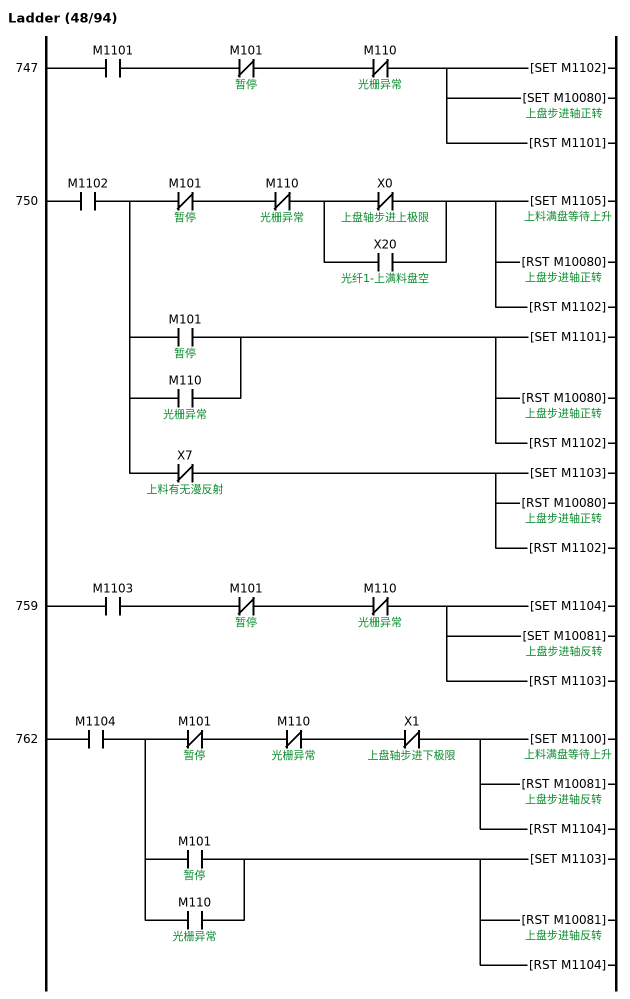
[picture p48: Ladder rows 747-762]
LD     M1101
ANI    M101	; 暂停
ANI    M110	; 光栅异常
SET    M1102
SET    M10080	; 上盘步进轴正转
RST    M1101
LD     M1102
MPS
ANI    M101	; 暂停
ANI    M110	; 光栅异常
LDI    X0	; 上盘轴步进上极限
OR     X20	; 光纤1-上满料盘空
ANB
SET    M1105	; 上料满盘等待上升
RST    M10080	; 上盘步进轴正转
RST    M1102
MRD
LD     M101	; 暂停
OR     M110	; 光栅异常
ANB
SET    M1101
RST    M10080	; 上盘步进轴正转
RST    M1102
MPP
ANI    X7	; 上料有无漫反射
SET    M1103
RST    M10080	; 上盘步进轴正转
RST    M1102
LD     M1103
ANI    M101	; 暂停
ANI    M110	; 光栅异常
SET    M1104
SET    M10081	; 上盘步进轴反转
RST    M1103
LD     M1104
MPS
ANI    M101	; 暂停
ANI    M110	; 光栅异常
ANI    X1	; 上盘轴步进下极限
SET    M1100	; 上料满盘等待上升
RST    M10081	; 上盘步进轴反转
RST    M1104
MPP
LD     M101	; 暂停
OR     M110	; 光栅异常
ANB
SET    M1103
RST    M10081	; 上盘步进轴反转
RST    M1104

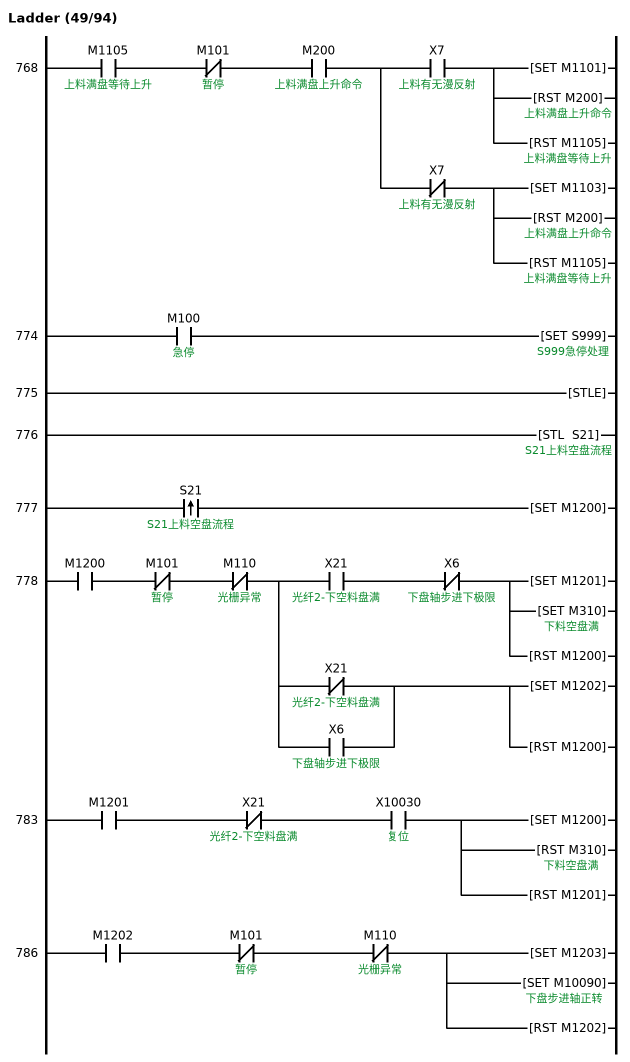
LD     M1105	; 上料满盘等待上升
ANI    M101	; 暂停
AND    M200	; 上料满盘上升命令
MPS
AND    X7	; 上料有无漫反射
SET    M1101
RST    M200	; 上料满盘上升命令
RST    M1105	; 上料满盘等待上升
MPP
ANI    X7	; 上料有无漫反射
SET    M1103
RST    M200	; 上料满盘上升命令
RST    M1105	; 上料满盘等待上升
LD     M100	; 急停
SET    S999	; S999急停处理
STLE
STL    S21	; S21上料空盘流程
LDP    S21	; S21上料空盘流程
SET    M1200
LD     M1200
ANI    M101	; 暂停
ANI    M110	; 光栅异常
MPS
AND    X21	; 光纤2-下空料盘满
ANI    X6	; 下盘轴步进下极限
SET    M1201
SET    M310	; 下料空盘满
RST    M1200
MPP
LDI    X21	; 光纤2-下空料盘满
OR     X6	; 下盘轴步进下极限
ANB
SET    M1202
RST    M1200
LD     M1201
ANI    X21	; 光纤2-下空料盘满
AND    X10030	; 复位
SET    M1200
RST    M310	; 下料空盘满
RST    M1201
LD     M1202
ANI    M101	; 暂停
ANI    M110	; 光栅异常
SET    M1203
SET    M10090	; 下盘步进轴正转
RST    M1202

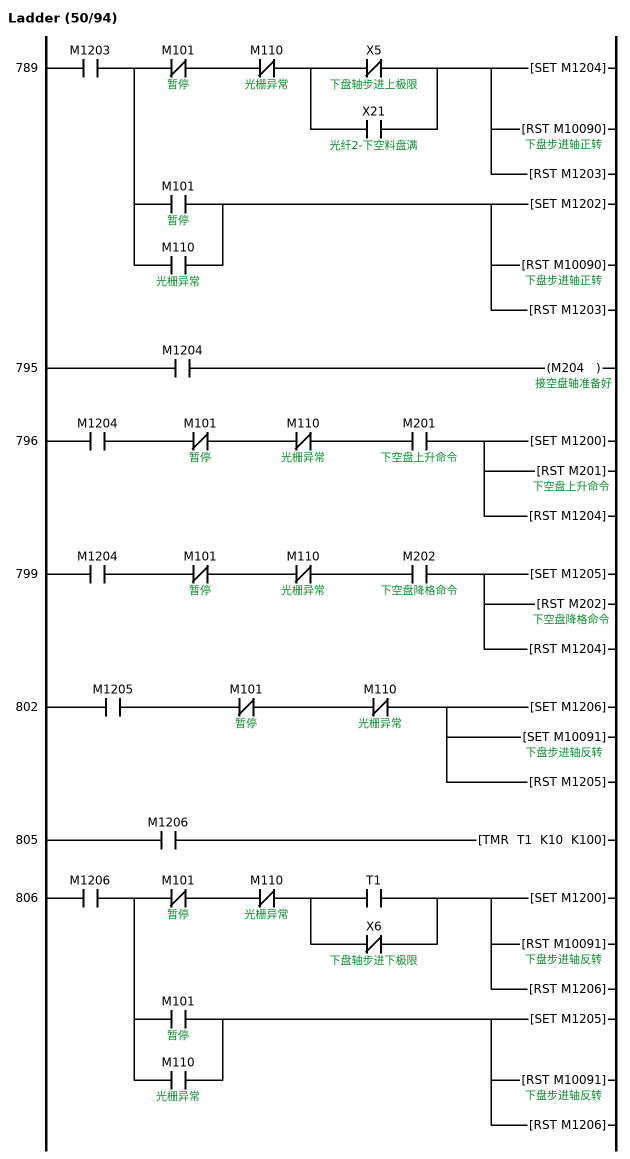
LD     M1203
MPS
ANI    M101	; 暂停
ANI    M110	; 光栅异常
LDI    X5	; 下盘轴步进上极限
OR     X21	; 光纤2-下空料盘满
ANB
SET    M1204
RST    M10090	; 下盘步进轴正转
RST    M1203
MPP
LD     M101	; 暂停
OR     M110	; 光栅异常
ANB
SET    M1202
RST    M10090	; 下盘步进轴正转
RST    M1203
LD     M1204
OUT    M204	; 接空盘轴准备好
LD     M1204
ANI    M101	; 暂停
ANI    M110	; 光栅异常
AND    M201	; 下空盘上升命令
SET    M1200
RST    M201	; 下空盘上升命令
RST    M1204
LD     M1204
ANI    M101	; 暂停
ANI    M110	; 光栅异常
AND    M202	; 下空盘降格命令
SET    M1205
RST    M202	; 下空盘降格命令
RST    M1204
LD     M1205
ANI    M101	; 暂停
ANI    M110	; 光栅异常
SET    M1206
SET    M10091	; 下盘步进轴反转
RST    M1205
LD     M1206
TMR    T1 K10 K100
LD     M1206
MPS
ANI    M101	; 暂停
ANI    M110	; 光栅异常
LD     T1
ORI    X6	; 下盘轴步进下极限
ANB
SET    M1200
RST    M10091	; 下盘步进轴反转
RST    M1206
MPP
LD     M101	; 暂停
OR     M110	; 光栅异常
ANB
SET    M1205
RST    M10091	; 下盘步进轴反转
RST    M1206

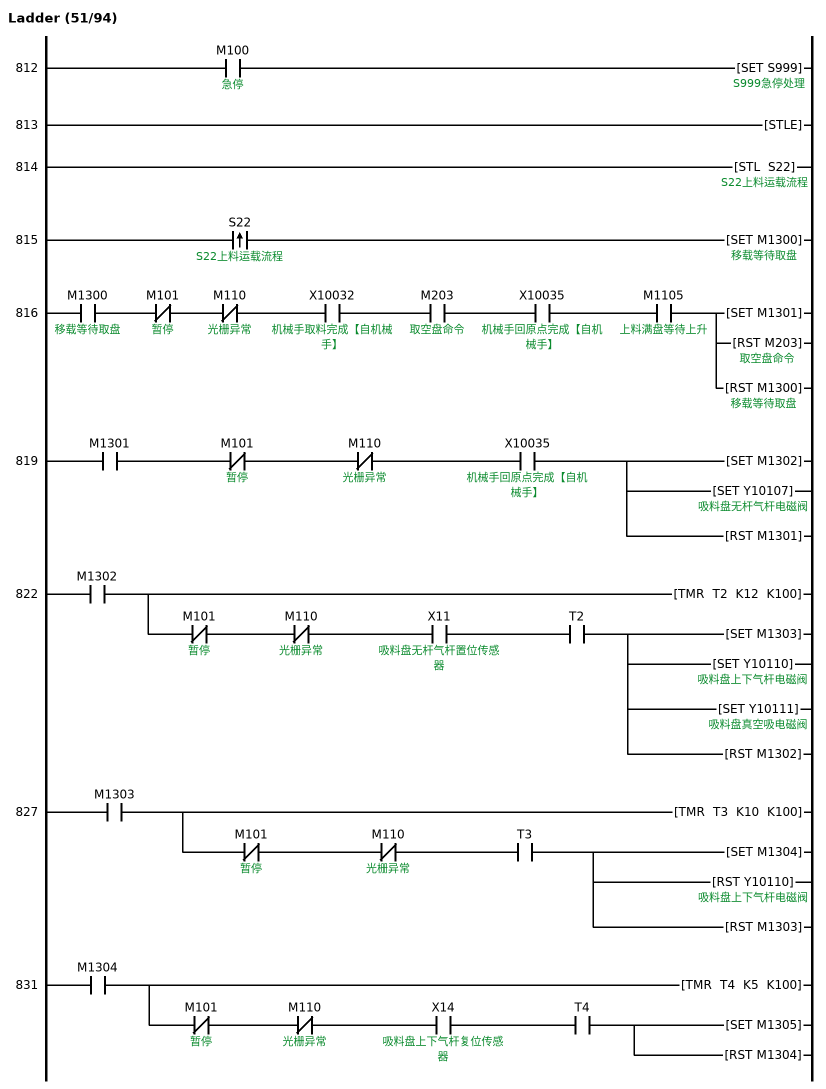
LD     M100	; 急停
SET    S999	; S999急停处理
STLE
STL    S22	; S22上料运载流程
LDP    S22	; S22上料运载流程
SET    M1300	; 移载等待取盘
LD     M1300	; 移载等待取盘
ANI    M101	; 暂停
ANI    M110	; 光栅异常
AND    X10032	; 机械手取料完成【自机械手】
AND    M203	; 取空盘命令
AND    X10035	; 机械手回原点完成【自机械手】
AND    M1105	; 上料满盘等待上升
SET    M1301
RST    M203	; 取空盘命令
RST    M1300	; 移载等待取盘
LD     M1301
ANI    M101	; 暂停
ANI    M110	; 光栅异常
AND    X10035	; 机械手回原点完成【自机械手】
SET    M1302
SET    Y10107	; 吸料盘无杆气杆电磁阀
RST    M1301
LD     M1302
TMR    T2 K12 K100
ANI    M101	; 暂停
ANI    M110	; 光栅异常
AND    X11	; 吸料盘无杆气杆置位传感器
AND    T2
SET    M1303
SET    Y10110	; 吸料盘上下气杆电磁阀
SET    Y10111	; 吸料盘真空吸电磁阀
RST    M1302
LD     M1303
TMR    T3 K10 K100
ANI    M101	; 暂停
ANI    M110	; 光栅异常
AND    T3
SET    M1304
RST    Y10110	; 吸料盘上下气杆电磁阀
RST    M1303
LD     M1304
TMR    T4 K5 K100
ANI    M101	; 暂停
ANI    M110	; 光栅异常
AND    X14	; 吸料盘上下气杆复位传感器
AND    T4
SET    M1305
RST    M1304

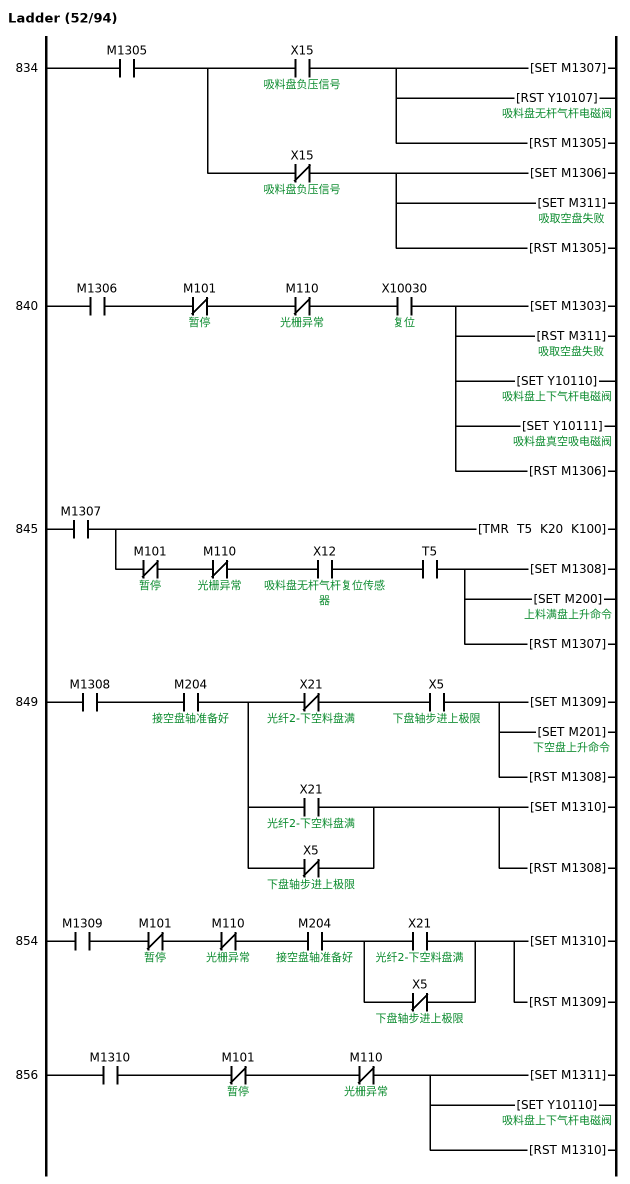
LD     M1305
MPS
AND    X15	; 吸料盘负压信号
SET    M1307
RST    Y10107	; 吸料盘无杆气杆电磁阀
RST    M1305
MPP
ANI    X15	; 吸料盘负压信号
SET    M1306
SET    M311	; 吸取空盘失败
RST    M1305
LD     M1306
ANI    M101	; 暂停
ANI    M110	; 光栅异常
AND    X10030	; 复位
SET    M1303
RST    M311	; 吸取空盘失败
SET    Y10110	; 吸料盘上下气杆电磁阀
SET    Y10111	; 吸料盘真空吸电磁阀
RST    M1306
LD     M1307
TMR    T5 K20 K100
ANI    M101	; 暂停
ANI    M110	; 光栅异常
AND    X12	; 吸料盘无杆气杆复位传感器
AND    T5
SET    M1308
SET    M200	; 上料满盘上升命令
RST    M1307
LD     M1308
AND    M204	; 接空盘轴准备好
MPS
ANI    X21	; 光纤2-下空料盘满
AND    X5	; 下盘轴步进上极限
SET    M1309
SET    M201	; 下空盘上升命令
RST    M1308
MPP
LD     X21	; 光纤2-下空料盘满
ORI    X5	; 下盘轴步进上极限
ANB
SET    M1310
RST    M1308
LD     M1309
ANI    M101	; 暂停
ANI    M110	; 光栅异常
AND    M204	; 接空盘轴准备好
LD     X21	; 光纤2-下空料盘满
ORI    X5	; 下盘轴步进上极限
ANB
SET    M1310
RST    M1309
LD     M1310
ANI    M101	; 暂停
ANI    M110	; 光栅异常
SET    M1311
SET    Y10110	; 吸料盘上下气杆电磁阀
RST    M1310

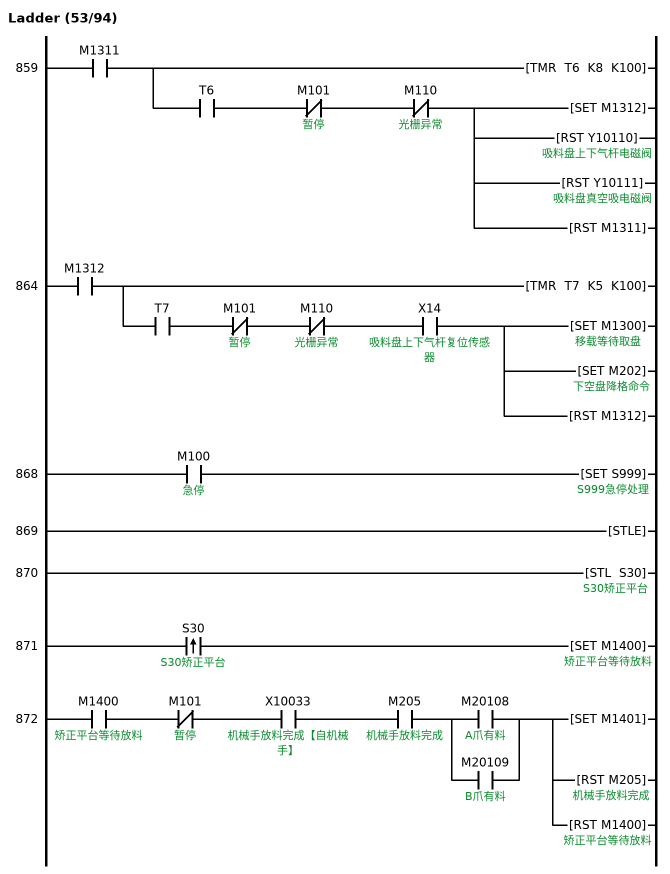
LD     M1311
TMR    T6 K8 K100
AND    T6
ANI    M101	; 暂停
ANI    M110	; 光栅异常
SET    M1312
RST    Y10110	; 吸料盘上下气杆电磁阀
RST    Y10111	; 吸料盘真空吸电磁阀
RST    M1311
LD     M1312
TMR    T7 K5 K100
AND    T7
ANI    M101	; 暂停
ANI    M110	; 光栅异常
AND    X14	; 吸料盘上下气杆复位传感器
SET    M1300	; 移载等待取盘
SET    M202	; 下空盘降格命令
RST    M1312
LD     M100	; 急停
SET    S999	; S999急停处理
STLE
STL    S30	; S30矫正平台
LDP    S30	; S30矫正平台
SET    M1400	; 矫正平台等待放料
LD     M1400	; 矫正平台等待放料
ANI    M101	; 暂停
AND    X10033	; 机械手放料完成【自机械手】
AND    M205	; 机械手放料完成
LD     M20108	; A爪有料
OR     M20109	; B爪有料
ANB
SET    M1401
RST    M205	; 机械手放料完成
RST    M1400	; 矫正平台等待放料

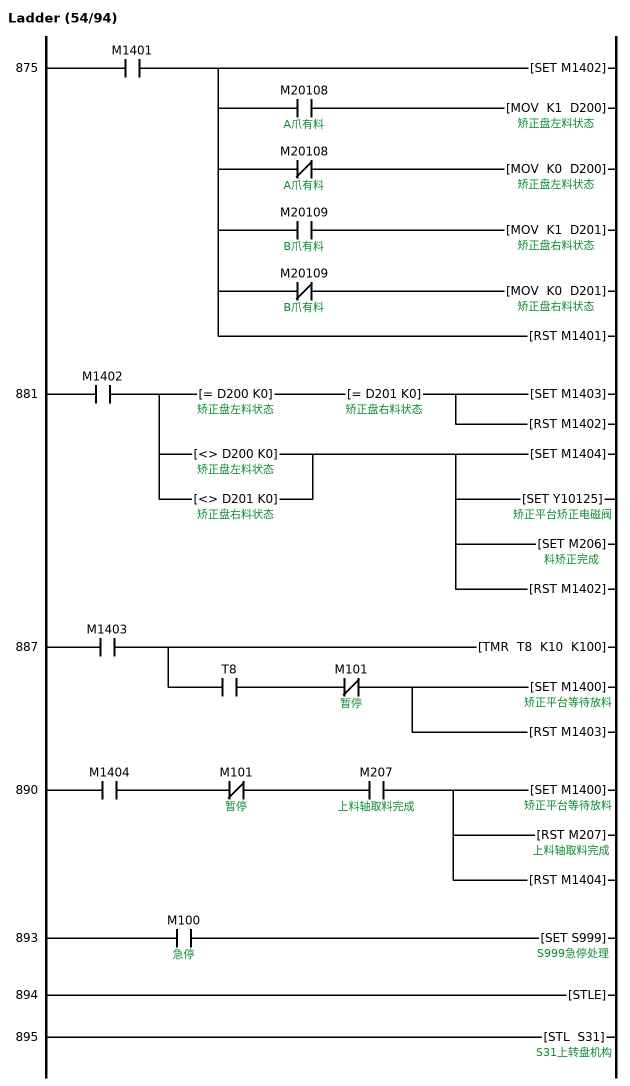
LD     M1401
SET    M1402
MPS
AND    M20108	; A爪有料
MOV    K1 D200	; 矫正盘左料状态
MRD
ANI    M20108	; A爪有料
MOV    K0 D200	; 矫正盘左料状态
MRD
AND    M20109	; B爪有料
MOV    K1 D201	; 矫正盘右料状态
MRD
ANI    M20109	; B爪有料
MOV    K0 D201	; 矫正盘右料状态
MPP
RST    M1401
LD     M1402
MPS
AND=   D200 K0	; 矫正盘左料状态
AND=   D201 K0	; 矫正盘右料状态
SET    M1403
RST    M1402
MPP
LD<>   D200 K0	; 矫正盘左料状态
OR<>   D201 K0	; 矫正盘右料状态
ANB
SET    M1404
SET    Y10125	; 矫正平台矫正电磁阀
SET    M206	; 料矫正完成
RST    M1402
LD     M1403
TMR    T8 K10 K100
AND    T8
ANI    M101	; 暂停
SET    M1400	; 矫正平台等待放料
RST    M1403
LD     M1404
ANI    M101	; 暂停
AND    M207	; 上料轴取料完成
SET    M1400	; 矫正平台等待放料
RST    M207	; 上料轴取料完成
RST    M1404
LD     M100	; 急停
SET    S999	; S999急停处理
STLE
STL    S31	; S31上转盘机构

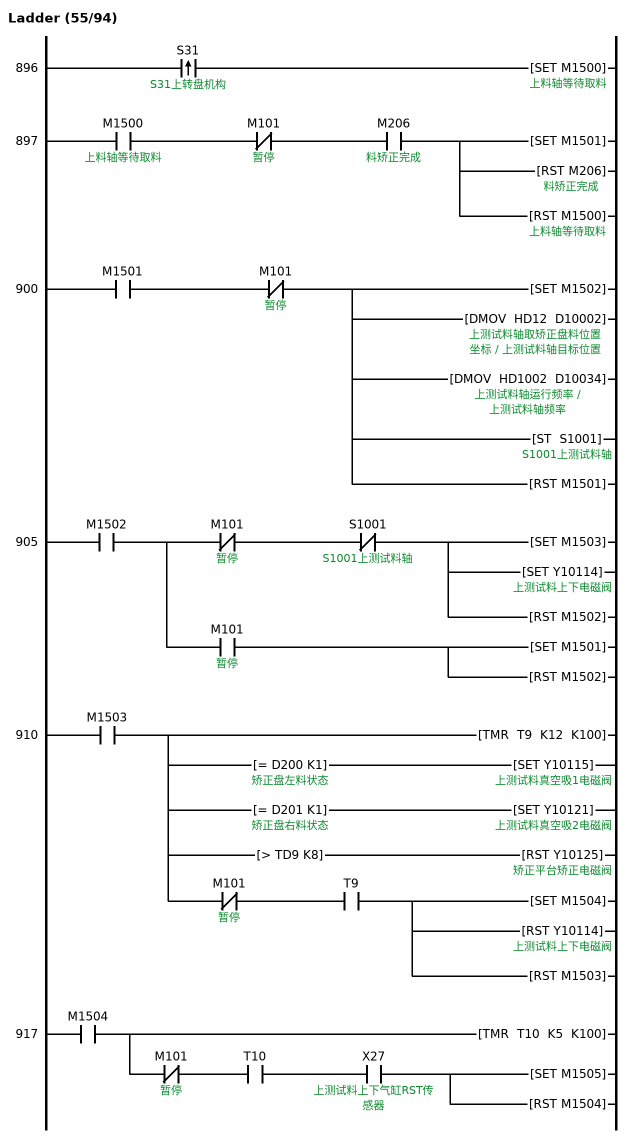
LDP    S31	; S31上转盘机构
SET    M1500	; 上料轴等待取料
LD     M1500	; 上料轴等待取料
ANI    M101	; 暂停
AND    M206	; 料矫正完成
SET    M1501
RST    M206	; 料矫正完成
RST    M1500	; 上料轴等待取料
LD     M1501
ANI    M101	; 暂停
SET    M1502
DMOV   HD12 D10002	; 上测试料轴取矫正盘料位置坐标 / 上测试料轴目标位置
DMOV   HD1002 D10034	; 上测试料轴运行频率 / 上测试料轴频率
ST     S1001	; S1001上测试料轴
RST    M1501
LD     M1502
MPS
ANI    M101	; 暂停
ANI    S1001	; S1001上测试料轴
SET    M1503
SET    Y10114	; 上测试料上下电磁阀
RST    M1502
MPP
AND    M101	; 暂停
SET    M1501
RST    M1502
LD     M1503
TMR    T9 K12 K100
MPS
AND=   D200 K1	; 矫正盘左料状态
SET    Y10115	; 上测试料真空吸1电磁阀
MRD
AND=   D201 K1	; 矫正盘右料状态
SET    Y10121	; 上测试料真空吸2电磁阀
MRD
AND>   TD9 K8
RST    Y10125	; 矫正平台矫正电磁阀
MPP
ANI    M101	; 暂停
AND    T9
SET    M1504
RST    Y10114	; 上测试料上下电磁阀
RST    M1503
LD     M1504
TMR    T10 K5 K100
ANI    M101	; 暂停
AND    T10
AND    X27	; 上测试料上下气缸RST传感器
SET    M1505
RST    M1504

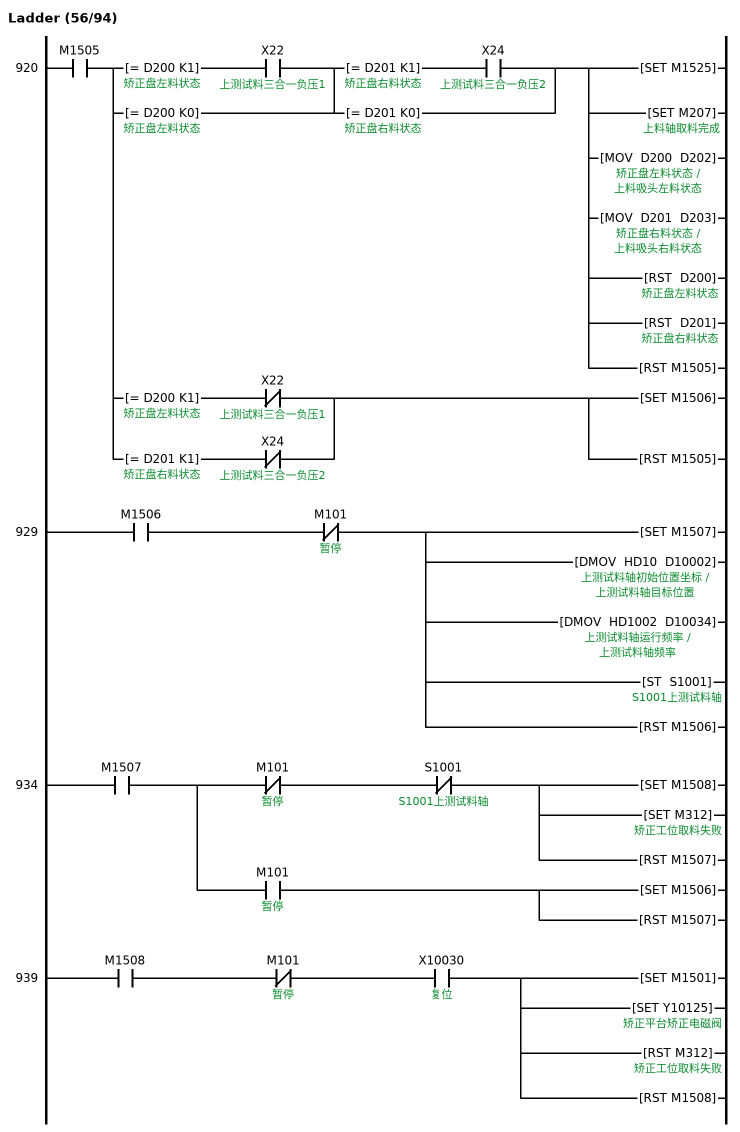
LD     M1505
MPS
LD=    D200 K1	; 矫正盘左料状态
AND    X22	; 上测试料三合一负压1
OR=    D200 K0	; 矫正盘左料状态
ANB
LD=    D201 K1	; 矫正盘右料状态
AND    X24	; 上测试料三合一负压2
OR=    D201 K0	; 矫正盘右料状态
ANB
SET    M1525
SET    M207	; 上料轴取料完成
MOV    D200 D202	; 矫正盘左料状态 / 上料吸头左料状态
MOV    D201 D203	; 矫正盘右料状态 / 上料吸头右料状态
RST    D200	; 矫正盘左料状态
RST    D201	; 矫正盘右料状态
RST    M1505
MPP
LD=    D200 K1	; 矫正盘左料状态
ANI    X22	; 上测试料三合一负压1
LD=    D201 K1	; 矫正盘右料状态
ANI    X24	; 上测试料三合一负压2
ORB
ANB
SET    M1506
RST    M1505
LD     M1506
ANI    M101	; 暂停
SET    M1507
DMOV   HD10 D10002	; 上测试料轴初始位置坐标 / 上测试料轴目标位置
DMOV   HD1002 D10034	; 上测试料轴运行频率 / 上测试料轴频率
ST     S1001	; S1001上测试料轴
RST    M1506
LD     M1507
MPS
ANI    M101	; 暂停
ANI    S1001	; S1001上测试料轴
SET    M1508
SET    M312	; 矫正工位取料失败
RST    M1507
MPP
AND    M101	; 暂停
SET    M1506
RST    M1507
LD     M1508
ANI    M101	; 暂停
AND    X10030	; 复位
SET    M1501
SET    Y10125	; 矫正平台矫正电磁阀
RST    M312	; 矫正工位取料失败
RST    M1508

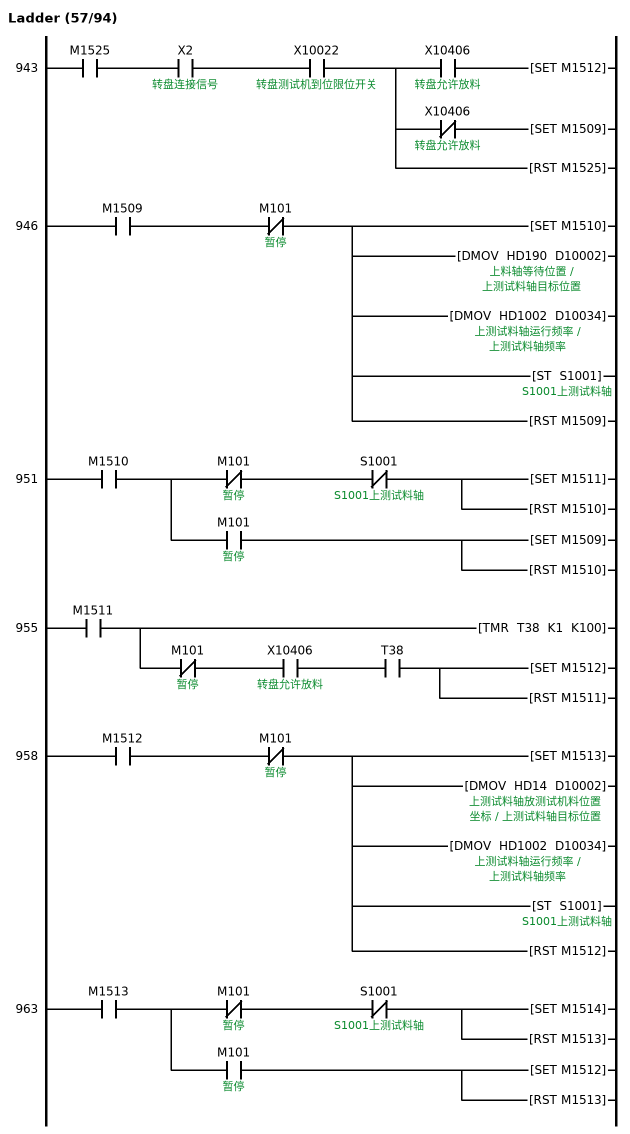
LD     M1525
AND    X2	; 转盘连接信号
AND    X10022	; 转盘测试机到位限位开关
MPS
AND    X10406	; 转盘允许放料
SET    M1512
MRD
ANI    X10406	; 转盘允许放料
SET    M1509
MPP
RST    M1525
LD     M1509
ANI    M101	; 暂停
SET    M1510
DMOV   HD190 D10002	; 上料轴等待位置 / 上测试料轴目标位置
DMOV   HD1002 D10034	; 上测试料轴运行频率 / 上测试料轴频率
ST     S1001	; S1001上测试料轴
RST    M1509
LD     M1510
MPS
ANI    M101	; 暂停
ANI    S1001	; S1001上测试料轴
SET    M1511
RST    M1510
MPP
AND    M101	; 暂停
SET    M1509
RST    M1510
LD     M1511
TMR    T38 K1 K100
ANI    M101	; 暂停
AND    X10406	; 转盘允许放料
AND    T38
SET    M1512
RST    M1511
LD     M1512
ANI    M101	; 暂停
SET    M1513
DMOV   HD14 D10002	; 上测试料轴放测试机料位置坐标 / 上测试料轴目标位置
DMOV   HD1002 D10034	; 上测试料轴运行频率 / 上测试料轴频率
ST     S1001	; S1001上测试料轴
RST    M1512
LD     M1513
MPS
ANI    M101	; 暂停
ANI    S1001	; S1001上测试料轴
SET    M1514
RST    M1513
MPP
AND    M101	; 暂停
SET    M1512
RST    M1513

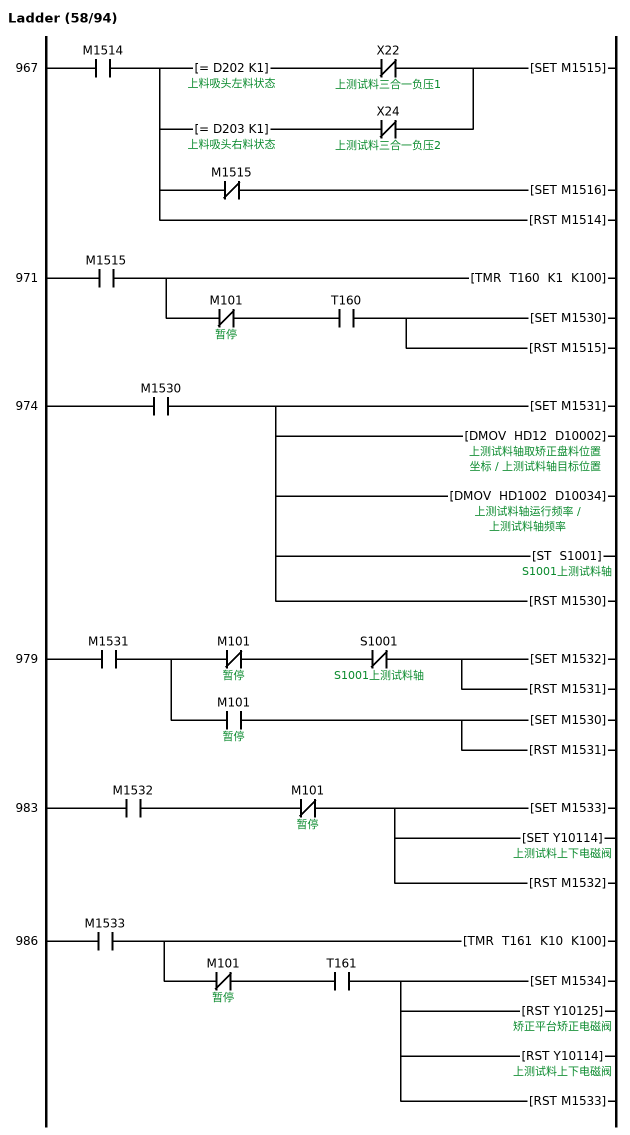
LD     M1514
MPS
LD=    D202 K1	; 上料吸头左料状态
ANI    X22	; 上测试料三合一负压1
LD=    D203 K1	; 上料吸头右料状态
ANI    X24	; 上测试料三合一负压2
ORB
ANB
SET    M1515
MRD
ANI    M1515
SET    M1516
MPP
RST    M1514
LD     M1515
TMR    T160 K1 K100
ANI    M101	; 暂停
AND    T160
SET    M1530
RST    M1515
LD     M1530
SET    M1531
DMOV   HD12 D10002	; 上测试料轴取矫正盘料位置坐标 / 上测试料轴目标位置
DMOV   HD1002 D10034	; 上测试料轴运行频率 / 上测试料轴频率
ST     S1001	; S1001上测试料轴
RST    M1530
LD     M1531
MPS
ANI    M101	; 暂停
ANI    S1001	; S1001上测试料轴
SET    M1532
RST    M1531
MPP
AND    M101	; 暂停
SET    M1530
RST    M1531
LD     M1532
ANI    M101	; 暂停
SET    M1533
SET    Y10114	; 上测试料上下电磁阀
RST    M1532
LD     M1533
TMR    T161 K10 K100
ANI    M101	; 暂停
AND    T161
SET    M1534
RST    Y10125	; 矫正平台矫正电磁阀
RST    Y10114	; 上测试料上下电磁阀
RST    M1533

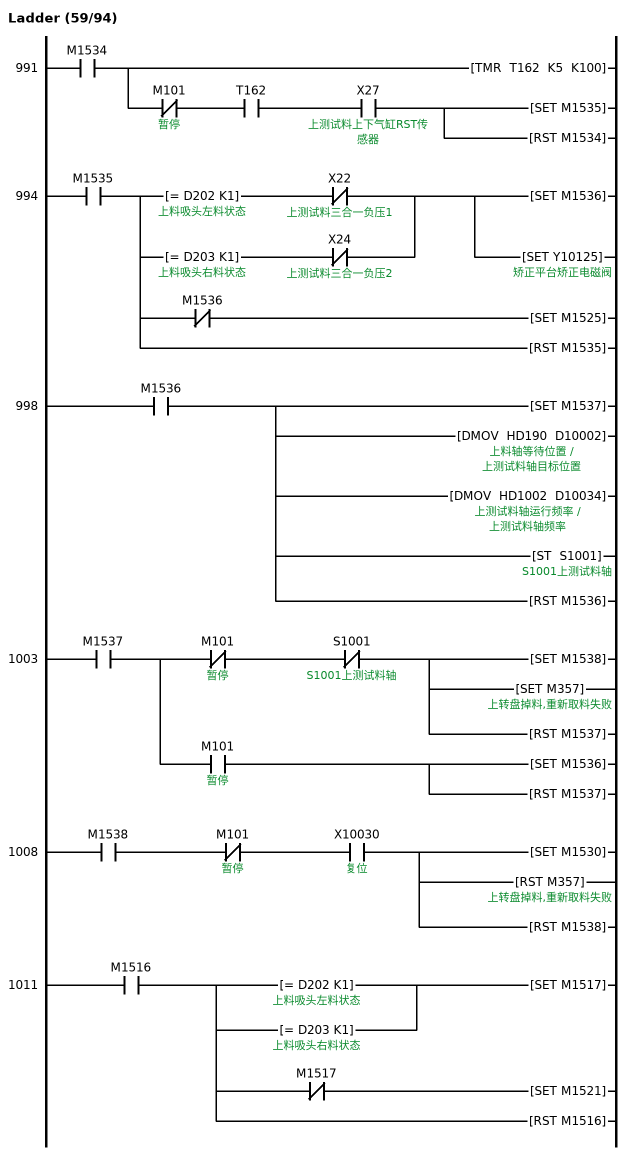
LD     M1534
TMR    T162 K5 K100
ANI    M101	; 暂停
AND    T162
AND    X27	; 上测试料上下气缸RST传感器
SET    M1535
RST    M1534
LD     M1535
MPS
LD=    D202 K1	; 上料吸头左料状态
ANI    X22	; 上测试料三合一负压1
LD=    D203 K1	; 上料吸头右料状态
ANI    X24	; 上测试料三合一负压2
ORB
ANB
SET    M1536
SET    Y10125	; 矫正平台矫正电磁阀
MRD
ANI    M1536
SET    M1525
MPP
RST    M1535
LD     M1536
SET    M1537
DMOV   HD190 D10002	; 上料轴等待位置 / 上测试料轴目标位置
DMOV   HD1002 D10034	; 上测试料轴运行频率 / 上测试料轴频率
ST     S1001	; S1001上测试料轴
RST    M1536
LD     M1537
MPS
ANI    M101	; 暂停
ANI    S1001	; S1001上测试料轴
SET    M1538
SET    M357	; 上转盘掉料,重新取料失败
RST    M1537
MPP
AND    M101	; 暂停
SET    M1536
RST    M1537
LD     M1538
ANI    M101	; 暂停
AND    X10030	; 复位
SET    M1530
RST    M357	; 上转盘掉料,重新取料失败
RST    M1538
LD     M1516
MPS
LD=    D202 K1	; 上料吸头左料状态
OR=    D203 K1	; 上料吸头右料状态
ANB
SET    M1517
MRD
ANI    M1517
SET    M1521
MPP
RST    M1516

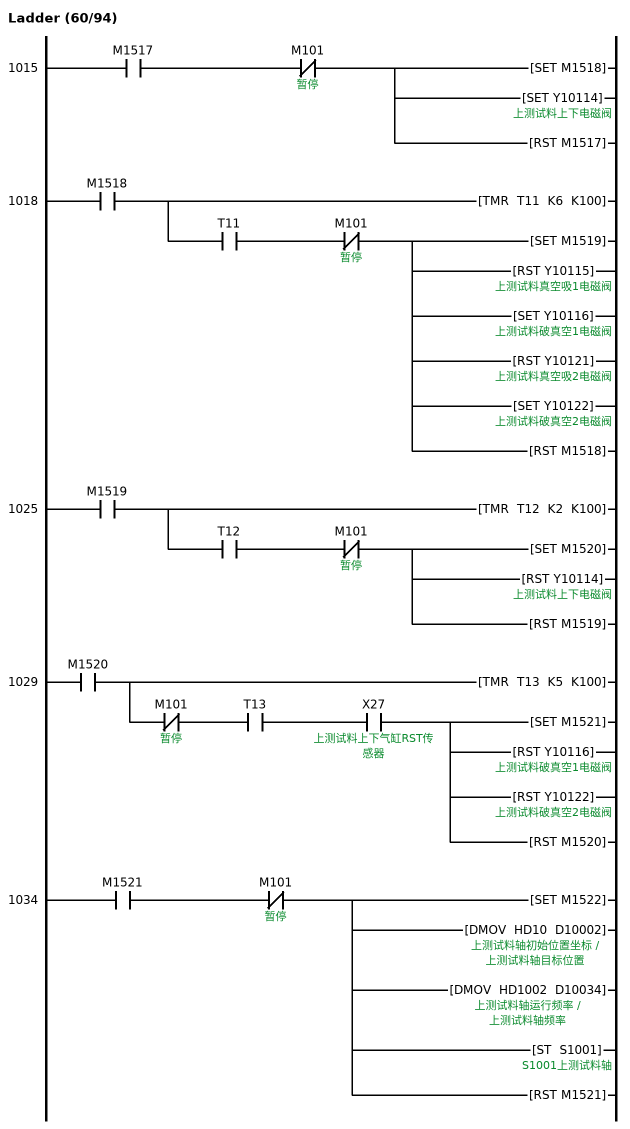
LD     M1517
ANI    M101	; 暂停
SET    M1518
SET    Y10114	; 上测试料上下电磁阀
RST    M1517
LD     M1518
TMR    T11 K6 K100
AND    T11
ANI    M101	; 暂停
SET    M1519
RST    Y10115	; 上测试料真空吸1电磁阀
SET    Y10116	; 上测试料破真空1电磁阀
RST    Y10121	; 上测试料真空吸2电磁阀
SET    Y10122	; 上测试料破真空2电磁阀
RST    M1518
LD     M1519
TMR    T12 K2 K100
AND    T12
ANI    M101	; 暂停
SET    M1520
RST    Y10114	; 上测试料上下电磁阀
RST    M1519
LD     M1520
TMR    T13 K5 K100
ANI    M101	; 暂停
AND    T13
AND    X27	; 上测试料上下气缸RST传感器
SET    M1521
RST    Y10116	; 上测试料破真空1电磁阀
RST    Y10122	; 上测试料破真空2电磁阀
RST    M1520
LD     M1521
ANI    M101	; 暂停
SET    M1522
DMOV   HD10 D10002	; 上测试料轴初始位置坐标 / 上测试料轴目标位置
DMOV   HD1002 D10034	; 上测试料轴运行频率 / 上测试料轴频率
ST     S1001	; S1001上测试料轴
RST    M1521

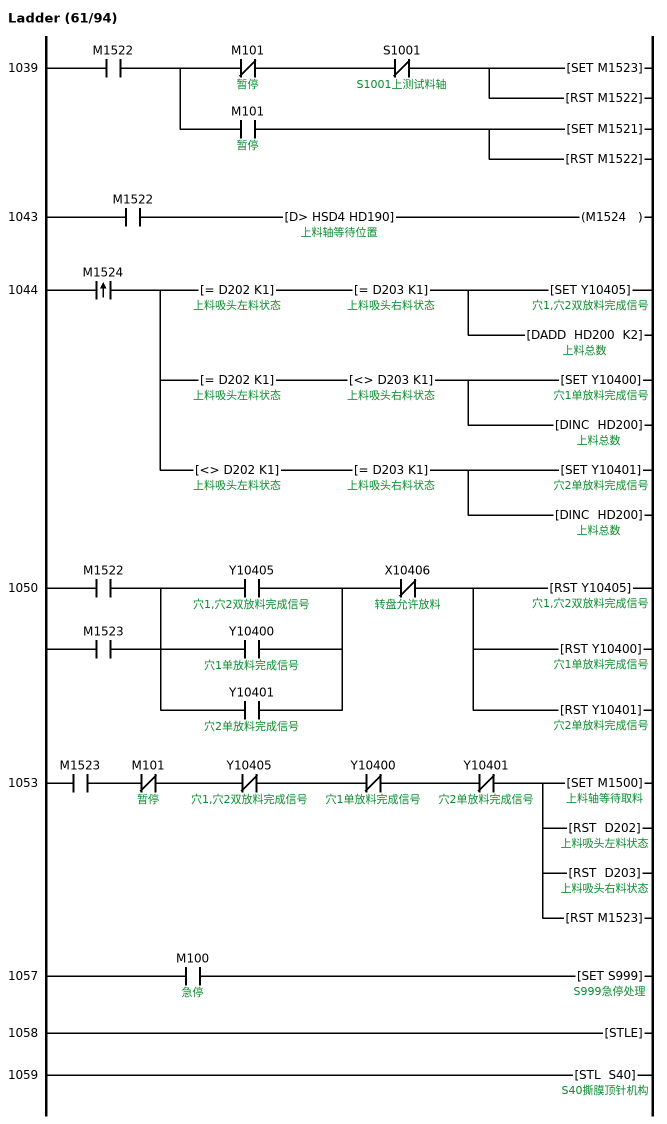
LD     M1522
MPS
ANI    M101	; 暂停
ANI    S1001	; S1001上测试料轴
SET    M1523
RST    M1522
MPP
AND    M101	; 暂停
SET    M1521
RST    M1522
LD     M1522
DAND>  HSD4 HD190	; 上料轴等待位置
OUT    M1524
LDP    M1524
MPS
AND=   D202 K1	; 上料吸头左料状态
AND=   D203 K1	; 上料吸头右料状态
SET    Y10405	; 穴1,穴2双放料完成信号
DADD   HD200 K2	; 上料总数
MRD
AND=   D202 K1	; 上料吸头左料状态
AND<>  D203 K1	; 上料吸头右料状态
SET    Y10400	; 穴1单放料完成信号
DINC   HD200	; 上料总数
MPP
AND<>  D202 K1	; 上料吸头左料状态
AND=   D203 K1	; 上料吸头右料状态
SET    Y10401	; 穴2单放料完成信号
DINC   HD200	; 上料总数
LD     M1522
OR     M1523
LD     Y10405	; 穴1,穴2双放料完成信号
OR     Y10400	; 穴1单放料完成信号
OR     Y10401	; 穴2单放料完成信号
ANB
ANI    X10406	; 转盘允许放料
RST    Y10405	; 穴1,穴2双放料完成信号
RST    Y10400	; 穴1单放料完成信号
RST    Y10401	; 穴2单放料完成信号
LD     M1523
ANI    M101	; 暂停
ANI    Y10405	; 穴1,穴2双放料完成信号
ANI    Y10400	; 穴1单放料完成信号
ANI    Y10401	; 穴2单放料完成信号
SET    M1500	; 上料轴等待取料
RST    D202	; 上料吸头左料状态
RST    D203	; 上料吸头右料状态
RST    M1523
LD     M100	; 急停
SET    S999	; S999急停处理
STLE
STL    S40	; S40撕膜顶针机构

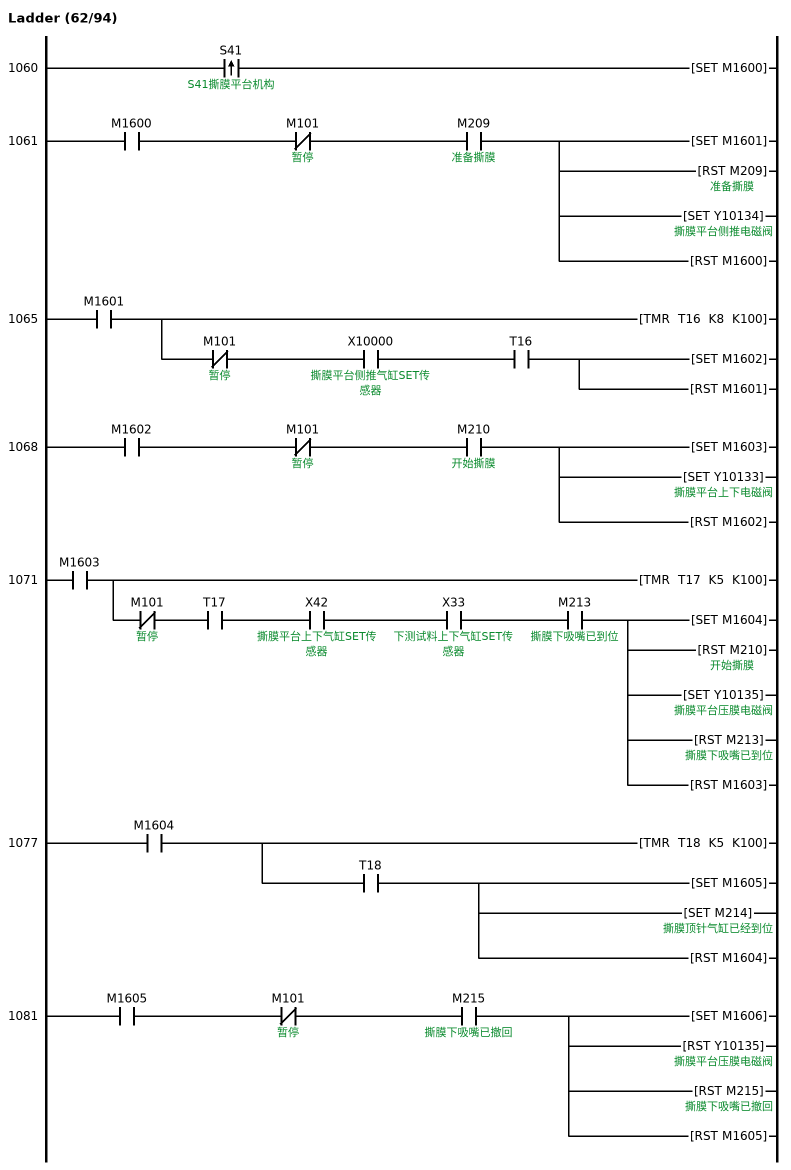
LDP    S41	; S41撕膜平台机构
SET    M1600
LD     M1600
ANI    M101	; 暂停
AND    M209	; 准备撕膜
SET    M1601
RST    M209	; 准备撕膜
SET    Y10134	; 撕膜平台侧推电磁阀
RST    M1600
LD     M1601
TMR    T16 K8 K100
ANI    M101	; 暂停
AND    X10000	; 撕膜平台侧推气缸SET传感器
AND    T16
SET    M1602
RST    M1601
LD     M1602
ANI    M101	; 暂停
AND    M210	; 开始撕膜
SET    M1603
SET    Y10133	; 撕膜平台上下电磁阀
RST    M1602
LD     M1603
TMR    T17 K5 K100
ANI    M101	; 暂停
AND    T17
AND    X42	; 撕膜平台上下气缸SET传感器
AND    X33	; 下测试料上下气缸SET传感器
AND    M213	; 撕膜下吸嘴已到位
SET    M1604
RST    M210	; 开始撕膜
SET    Y10135	; 撕膜平台压膜电磁阀
RST    M213	; 撕膜下吸嘴已到位
RST    M1603
LD     M1604
TMR    T18 K5 K100
AND    T18
SET    M1605
SET    M214	; 撕膜顶针气缸已经到位
RST    M1604
LD     M1605
ANI    M101	; 暂停
AND    M215	; 撕膜下吸嘴已撤回
SET    M1606
RST    Y10135	; 撕膜平台压膜电磁阀
RST    M215	; 撕膜下吸嘴已撤回
RST    M1605

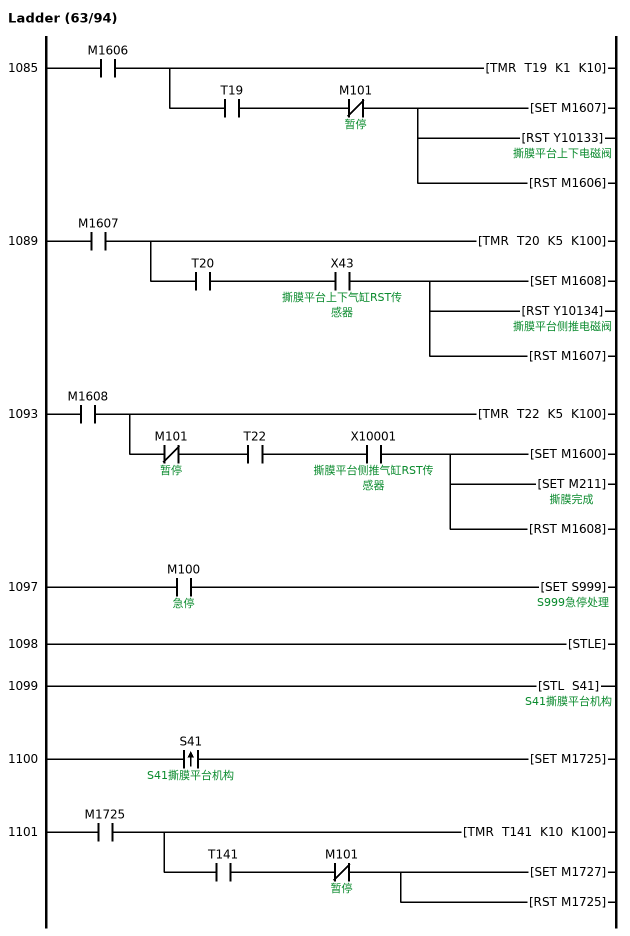
LD     M1606
TMR    T19 K1 K10
AND    T19
ANI    M101	; 暂停
SET    M1607
RST    Y10133	; 撕膜平台上下电磁阀
RST    M1606
LD     M1607
TMR    T20 K5 K100
AND    T20
AND    X43	; 撕膜平台上下气缸RST传感器
SET    M1608
RST    Y10134	; 撕膜平台侧推电磁阀
RST    M1607
LD     M1608
TMR    T22 K5 K100
ANI    M101	; 暂停
AND    T22
AND    X10001	; 撕膜平台侧推气缸RST传感器
SET    M1600
SET    M211	; 撕膜完成
RST    M1608
LD     M100	; 急停
SET    S999	; S999急停处理
STLE
STL    S41	; S41撕膜平台机构
LDP    S41	; S41撕膜平台机构
SET    M1725
LD     M1725
TMR    T141 K10 K100
AND    T141
ANI    M101	; 暂停
SET    M1727
RST    M1725

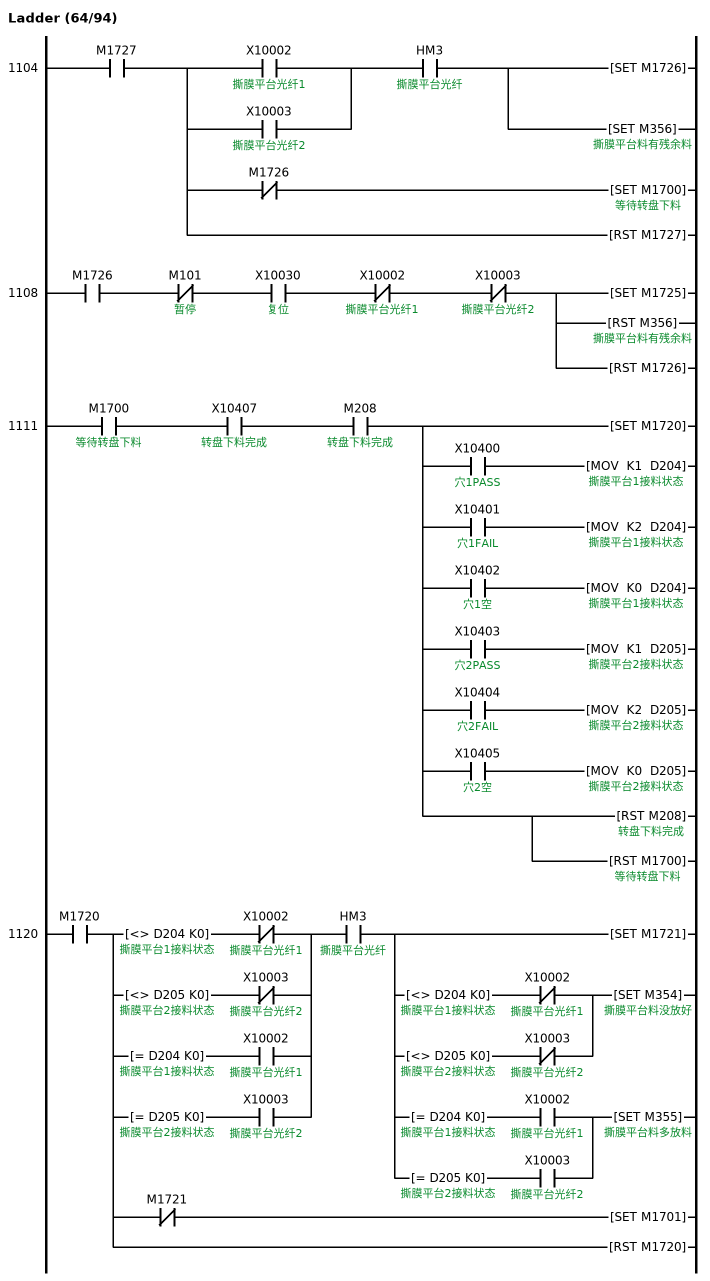
LD     M1727
MPS
LD     X10002	; 撕膜平台光纤1
OR     X10003	; 撕膜平台光纤2
ANB
AND    HM3	; 撕膜平台光纤
SET    M1726
SET    M356	; 撕膜平台料有残余料
MRD
ANI    M1726
SET    M1700	; 等待转盘下料
MPP
RST    M1727
LD     M1726
ANI    M101	; 暂停
AND    X10030	; 复位
ANI    X10002	; 撕膜平台光纤1
ANI    X10003	; 撕膜平台光纤2
SET    M1725
RST    M356	; 撕膜平台料有残余料
RST    M1726
LD     M1700	; 等待转盘下料
AND    X10407	; 转盘下料完成
AND    M208	; 转盘下料完成
SET    M1720
MPS
AND    X10400	; 穴1PASS
MOV    K1 D204	; 撕膜平台1接料状态
MRD
AND    X10401	; 穴1FAIL
MOV    K2 D204	; 撕膜平台1接料状态
MRD
AND    X10402	; 穴1空
MOV    K0 D204	; 撕膜平台1接料状态
MRD
AND    X10403	; 穴2PASS
MOV    K1 D205	; 撕膜平台2接料状态
MRD
AND    X10404	; 穴2FAIL
MOV    K2 D205	; 撕膜平台2接料状态
MRD
AND    X10405	; 穴2空
MOV    K0 D205	; 撕膜平台2接料状态
MPP
RST    M208	; 转盘下料完成
RST    M1700	; 等待转盘下料
LD     M1720
MPS
LD<>   D204 K0	; 撕膜平台1接料状态
ANI    X10002	; 撕膜平台光纤1
LD<>   D205 K0	; 撕膜平台2接料状态
ANI    X10003	; 撕膜平台光纤2
ORB
LD=    D204 K0	; 撕膜平台1接料状态
AND    X10002	; 撕膜平台光纤1
ORB
LD=    D205 K0	; 撕膜平台2接料状态
AND    X10003	; 撕膜平台光纤2
ORB
ANB
AND    HM3	; 撕膜平台光纤
SET    M1721
MPS
LD<>   D204 K0	; 撕膜平台1接料状态
ANI    X10002	; 撕膜平台光纤1
LD<>   D205 K0	; 撕膜平台2接料状态
ANI    X10003	; 撕膜平台光纤2
ORB
ANB
SET    M354	; 撕膜平台料没放好
MPP
LD=    D204 K0	; 撕膜平台1接料状态
AND    X10002	; 撕膜平台光纤1
LD=    D205 K0	; 撕膜平台2接料状态
AND    X10003	; 撕膜平台光纤2
ORB
ANB
SET    M355	; 撕膜平台料多放料
MRD
ANI    M1721
SET    M1701
MPP
RST    M1720

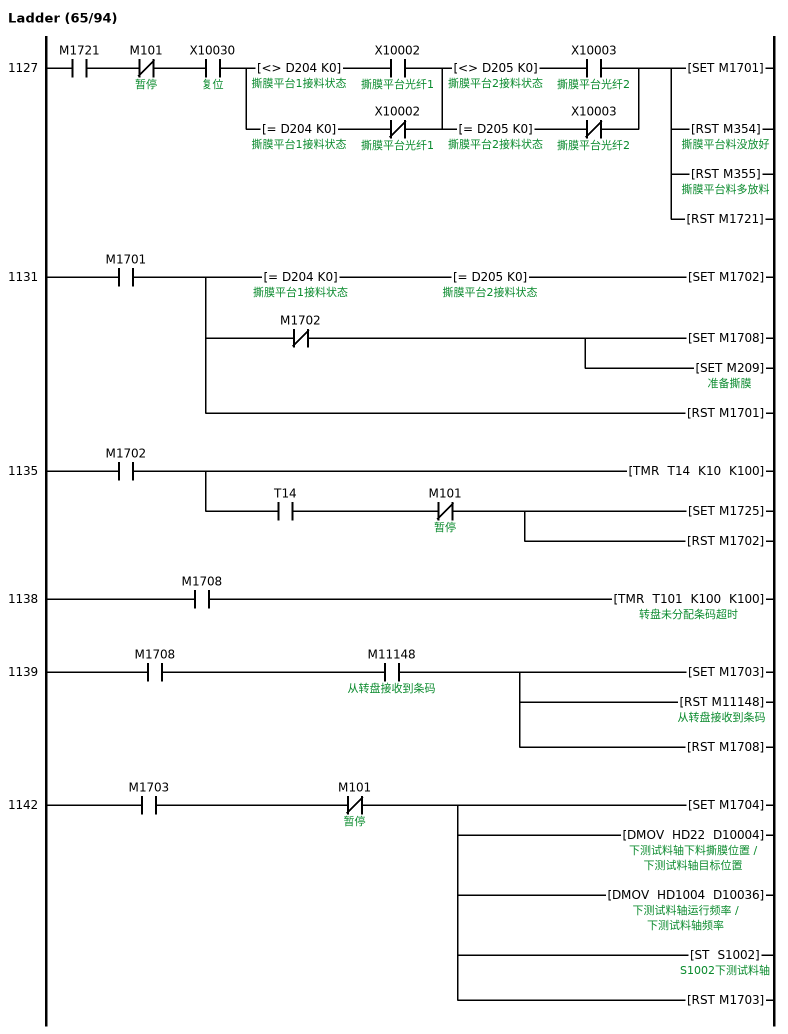
LD     M1721
ANI    M101	; 暂停
AND    X10030	; 复位
LD<>   D204 K0	; 撕膜平台1接料状态
AND    X10002	; 撕膜平台光纤1
LD=    D204 K0	; 撕膜平台1接料状态
ANI    X10002	; 撕膜平台光纤1
ORB
ANB
LD<>   D205 K0	; 撕膜平台2接料状态
AND    X10003	; 撕膜平台光纤2
LD=    D205 K0	; 撕膜平台2接料状态
ANI    X10003	; 撕膜平台光纤2
ORB
ANB
SET    M1701
RST    M354	; 撕膜平台料没放好
RST    M355	; 撕膜平台料多放料
RST    M1721
LD     M1701
MPS
AND=   D204 K0	; 撕膜平台1接料状态
AND=   D205 K0	; 撕膜平台2接料状态
SET    M1702
MRD
ANI    M1702
SET    M1708
SET    M209	; 准备撕膜
MPP
RST    M1701
LD     M1702
TMR    T14 K10 K100
AND    T14
ANI    M101	; 暂停
SET    M1725
RST    M1702
LD     M1708
TMR    T101 K100 K100	; 转盘未分配条码超时
LD     M1708
AND    M11148	; 从转盘接收到条码
SET    M1703
RST    M11148	; 从转盘接收到条码
RST    M1708
LD     M1703
ANI    M101	; 暂停
SET    M1704
DMOV   HD22 D10004	; 下测试料轴下料撕膜位置 / 下测试料轴目标位置
DMOV   HD1004 D10036	; 下测试料轴运行频率 / 下测试料轴频率
ST     S1002	; S1002下测试料轴
RST    M1703

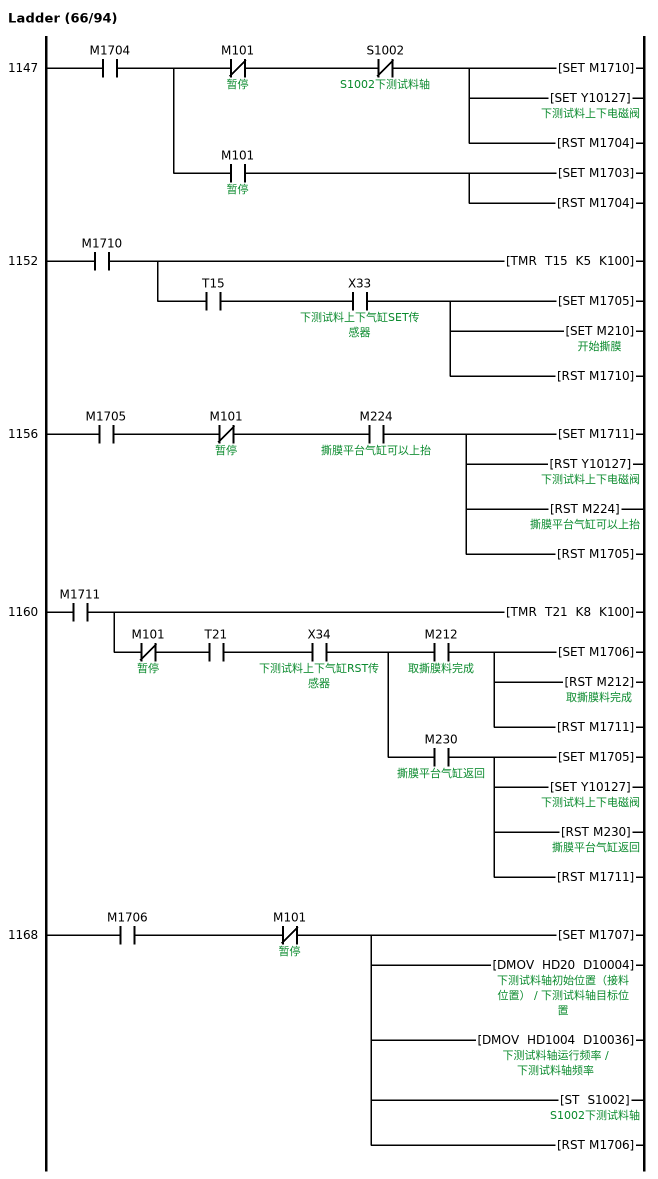
LD     M1704
MPS
ANI    M101	; 暂停
ANI    S1002	; S1002下测试料轴
SET    M1710
SET    Y10127	; 下测试料上下电磁阀
RST    M1704
MPP
AND    M101	; 暂停
SET    M1703
RST    M1704
LD     M1710
TMR    T15 K5 K100
AND    T15
AND    X33	; 下测试料上下气缸SET传感器
SET    M1705
SET    M210	; 开始撕膜
RST    M1710
LD     M1705
ANI    M101	; 暂停
AND    M224	; 撕膜平台气缸可以上抬
SET    M1711
RST    Y10127	; 下测试料上下电磁阀
RST    M224	; 撕膜平台气缸可以上抬
RST    M1705
LD     M1711
TMR    T21 K8 K100
ANI    M101	; 暂停
AND    T21
AND    X34	; 下测试料上下气缸RST传感器
MPS
AND    M212	; 取撕膜料完成
SET    M1706
RST    M212	; 取撕膜料完成
RST    M1711
MPP
AND    M230	; 撕膜平台气缸返回
SET    M1705
SET    Y10127	; 下测试料上下电磁阀
RST    M230	; 撕膜平台气缸返回
RST    M1711
LD     M1706
ANI    M101	; 暂停
SET    M1707
DMOV   HD20 D10004	; 下测试料轴初始位置（接料位置） / 下测试料轴目标位置
DMOV   HD1004 D10036	; 下测试料轴运行频率 / 下测试料轴频率
ST     S1002	; S1002下测试料轴
RST    M1706

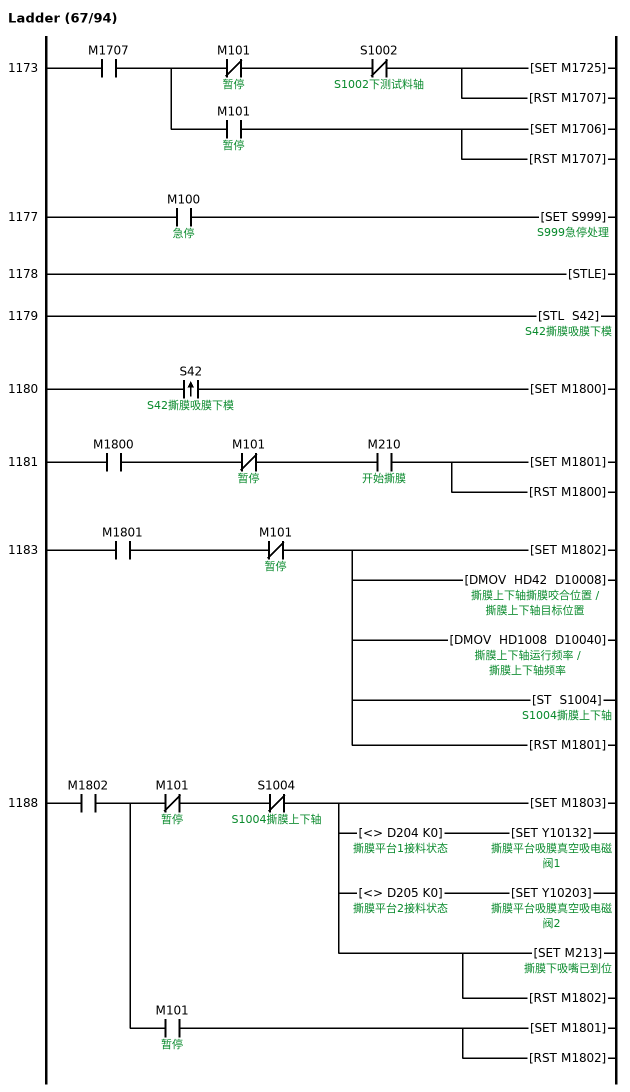
LD     M1707
MPS
ANI    M101	; 暂停
ANI    S1002	; S1002下测试料轴
SET    M1725
RST    M1707
MPP
AND    M101	; 暂停
SET    M1706
RST    M1707
LD     M100	; 急停
SET    S999	; S999急停处理
STLE
STL    S42	; S42撕膜吸膜下模
LDP    S42	; S42撕膜吸膜下模
SET    M1800
LD     M1800
ANI    M101	; 暂停
AND    M210	; 开始撕膜
SET    M1801
RST    M1800
LD     M1801
ANI    M101	; 暂停
SET    M1802
DMOV   HD42 D10008	; 撕膜上下轴撕膜咬合位置 / 撕膜上下轴目标位置
DMOV   HD1008 D10040	; 撕膜上下轴运行频率 / 撕膜上下轴频率
ST     S1004	; S1004撕膜上下轴
RST    M1801
LD     M1802
MPS
ANI    M101	; 暂停
ANI    S1004	; S1004撕膜上下轴
SET    M1803
MPS
AND<>  D204 K0	; 撕膜平台1接料状态
SET    Y10132	; 撕膜平台吸膜真空吸电磁阀1
MRD
AND<>  D205 K0	; 撕膜平台2接料状态
SET    Y10203	; 撕膜平台吸膜真空吸电磁阀2
MPP
SET    M213	; 撕膜下吸嘴已到位
RST    M1802
MPP
AND    M101	; 暂停
SET    M1801
RST    M1802

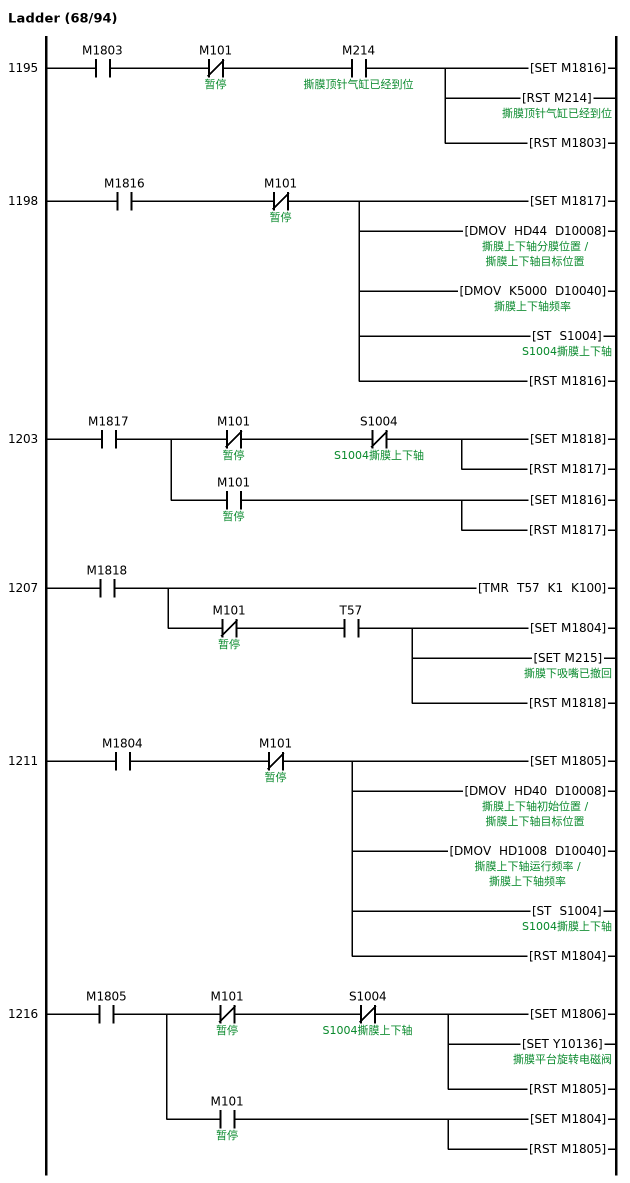
LD     M1803
ANI    M101	; 暂停
AND    M214	; 撕膜顶针气缸已经到位
SET    M1816
RST    M214	; 撕膜顶针气缸已经到位
RST    M1803
LD     M1816
ANI    M101	; 暂停
SET    M1817
DMOV   HD44 D10008	; 撕膜上下轴分膜位置 / 撕膜上下轴目标位置
DMOV   K5000 D10040	; 撕膜上下轴频率
ST     S1004	; S1004撕膜上下轴
RST    M1816
LD     M1817
MPS
ANI    M101	; 暂停
ANI    S1004	; S1004撕膜上下轴
SET    M1818
RST    M1817
MPP
AND    M101	; 暂停
SET    M1816
RST    M1817
LD     M1818
TMR    T57 K1 K100
ANI    M101	; 暂停
AND    T57
SET    M1804
SET    M215	; 撕膜下吸嘴已撤回
RST    M1818
LD     M1804
ANI    M101	; 暂停
SET    M1805
DMOV   HD40 D10008	; 撕膜上下轴初始位置 / 撕膜上下轴目标位置
DMOV   HD1008 D10040	; 撕膜上下轴运行频率 / 撕膜上下轴频率
ST     S1004	; S1004撕膜上下轴
RST    M1804
LD     M1805
MPS
ANI    M101	; 暂停
ANI    S1004	; S1004撕膜上下轴
SET    M1806
SET    Y10136	; 撕膜平台旋转电磁阀
RST    M1805
MPP
AND    M101	; 暂停
SET    M1804
RST    M1805

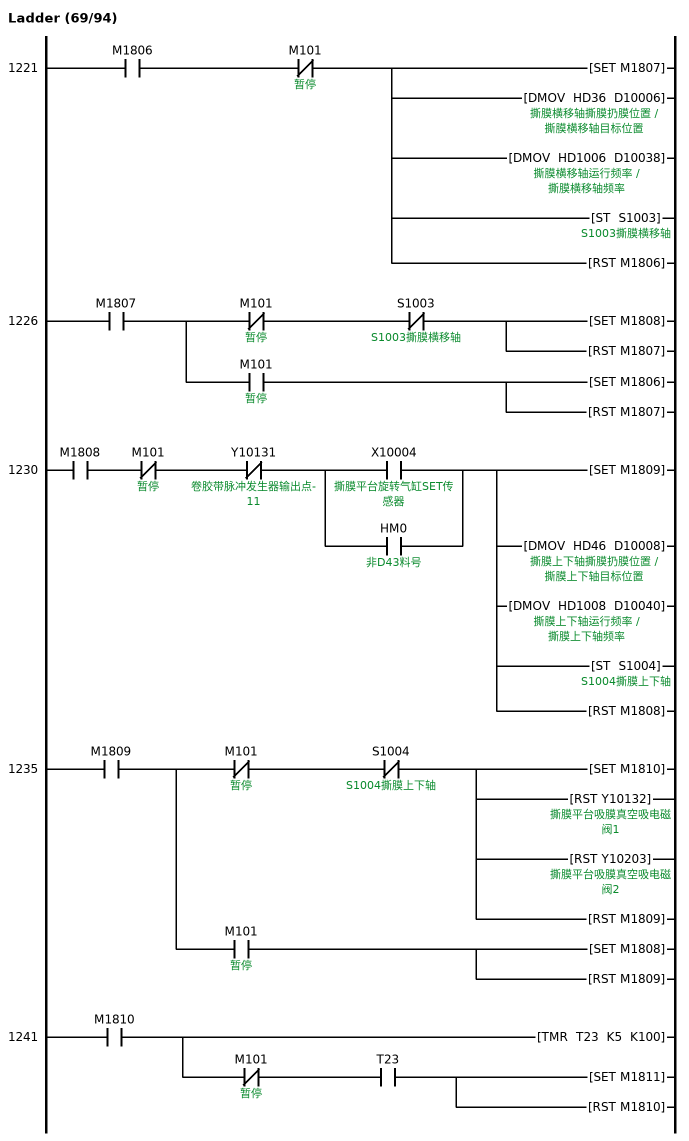
LD     M1806
ANI    M101	; 暂停
SET    M1807
DMOV   HD36 D10006	; 撕膜横移轴撕膜扔膜位置 / 撕膜横移轴目标位置
DMOV   HD1006 D10038	; 撕膜横移轴运行频率 / 撕膜横移轴频率
ST     S1003	; S1003撕膜横移轴
RST    M1806
LD     M1807
MPS
ANI    M101	; 暂停
ANI    S1003	; S1003撕膜横移轴
SET    M1808
RST    M1807
MPP
AND    M101	; 暂停
SET    M1806
RST    M1807
LD     M1808
ANI    M101	; 暂停
ANI    Y10131	; 卷胶带脉冲发生器输出点-11
LD     X10004	; 撕膜平台旋转气缸SET传感器
OR     HM0	; 非D43料号
ANB
SET    M1809
DMOV   HD46 D10008	; 撕膜上下轴撕膜扔膜位置 / 撕膜上下轴目标位置
DMOV   HD1008 D10040	; 撕膜上下轴运行频率 / 撕膜上下轴频率
ST     S1004	; S1004撕膜上下轴
RST    M1808
LD     M1809
MPS
ANI    M101	; 暂停
ANI    S1004	; S1004撕膜上下轴
SET    M1810
RST    Y10132	; 撕膜平台吸膜真空吸电磁阀1
RST    Y10203	; 撕膜平台吸膜真空吸电磁阀2
RST    M1809
MPP
AND    M101	; 暂停
SET    M1808
RST    M1809
LD     M1810
TMR    T23 K5 K100
ANI    M101	; 暂停
AND    T23
SET    M1811
RST    M1810

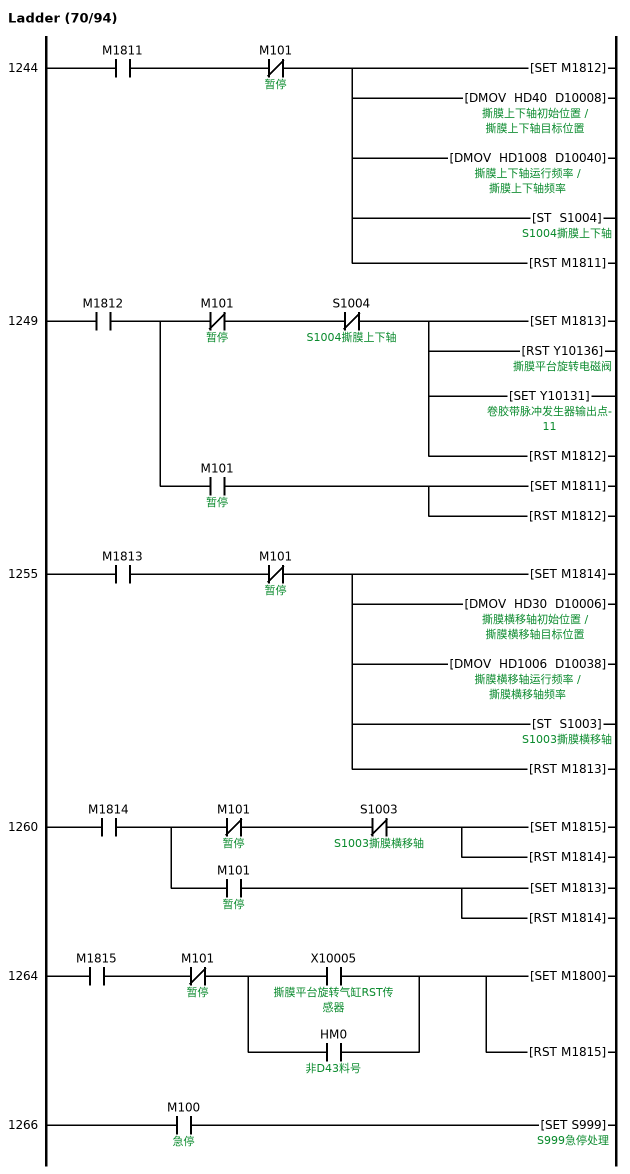
LD     M1811
ANI    M101	; 暂停
SET    M1812
DMOV   HD40 D10008	; 撕膜上下轴初始位置 / 撕膜上下轴目标位置
DMOV   HD1008 D10040	; 撕膜上下轴运行频率 / 撕膜上下轴频率
ST     S1004	; S1004撕膜上下轴
RST    M1811
LD     M1812
MPS
ANI    M101	; 暂停
ANI    S1004	; S1004撕膜上下轴
SET    M1813
RST    Y10136	; 撕膜平台旋转电磁阀
SET    Y10131	; 卷胶带脉冲发生器输出点-11
RST    M1812
MPP
AND    M101	; 暂停
SET    M1811
RST    M1812
LD     M1813
ANI    M101	; 暂停
SET    M1814
DMOV   HD30 D10006	; 撕膜横移轴初始位置 / 撕膜横移轴目标位置
DMOV   HD1006 D10038	; 撕膜横移轴运行频率 / 撕膜横移轴频率
ST     S1003	; S1003撕膜横移轴
RST    M1813
LD     M1814
MPS
ANI    M101	; 暂停
ANI    S1003	; S1003撕膜横移轴
SET    M1815
RST    M1814
MPP
AND    M101	; 暂停
SET    M1813
RST    M1814
LD     M1815
ANI    M101	; 暂停
LD     X10005	; 撕膜平台旋转气缸RST传感器
OR     HM0	; 非D43料号
ANB
SET    M1800
RST    M1815
LD     M100	; 急停
SET    S999	; S999急停处理

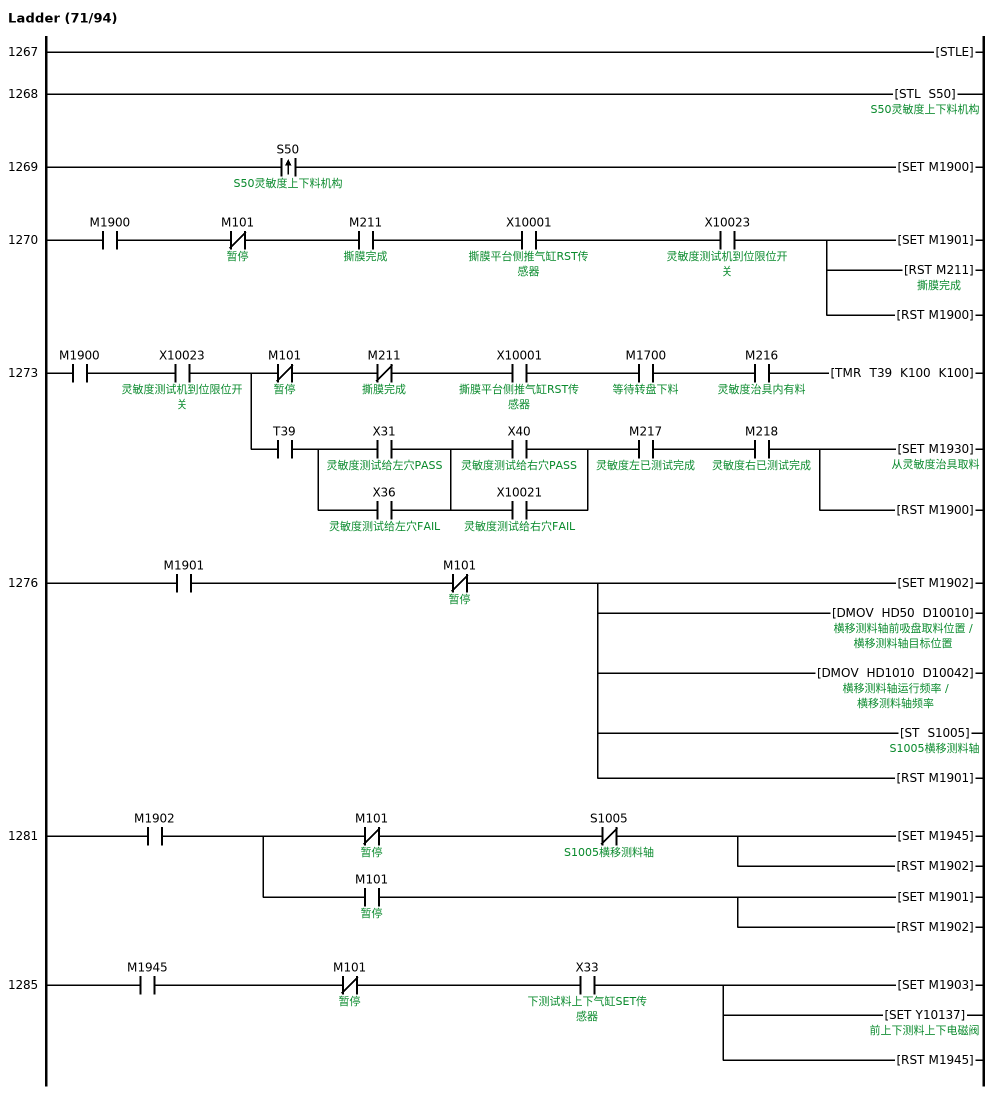
STLE
STL    S50	; S50灵敏度上下料机构
LDP    S50	; S50灵敏度上下料机构
SET    M1900
LD     M1900
ANI    M101	; 暂停
AND    M211	; 撕膜完成
AND    X10001	; 撕膜平台侧推气缸RST传感器
AND    X10023	; 灵敏度测试机到位限位开关
SET    M1901
RST    M211	; 撕膜完成
RST    M1900
LD     M1900
AND    X10023	; 灵敏度测试机到位限位开关
MPS
ANI    M101	; 暂停
ANI    M211	; 撕膜完成
AND    X10001	; 撕膜平台侧推气缸RST传感器
AND    M1700	; 等待转盘下料
AND    M216	; 灵敏度治具内有料
TMR    T39 K100 K100
MPP
AND    T39
LD     X31	; 灵敏度测试给左穴PASS
OR     X36	; 灵敏度测试给左穴FAIL
ANB
LD     X40	; 灵敏度测试给右穴PASS
OR     X10021	; 灵敏度测试给右穴FAIL
ANB
AND    M217	; 灵敏度左已测试完成
AND    M218	; 灵敏度右已测试完成
SET    M1930	; 从灵敏度治具取料
RST    M1900
LD     M1901
ANI    M101	; 暂停
SET    M1902
DMOV   HD50 D10010	; 横移测料轴前吸盘取料位置 / 横移测料轴目标位置
DMOV   HD1010 D10042	; 横移测料轴运行频率 / 横移测料轴频率
ST     S1005	; S1005横移测料轴
RST    M1901
LD     M1902
MPS
ANI    M101	; 暂停
ANI    S1005	; S1005横移测料轴
SET    M1945
RST    M1902
MPP
AND    M101	; 暂停
SET    M1901
RST    M1902
LD     M1945
ANI    M101	; 暂停
AND    X33	; 下测试料上下气缸SET传感器
SET    M1903
SET    Y10137	; 前上下测料上下电磁阀
RST    M1945

